// TwinCAT 3 PLC project PLC
// ProgramVersion: 3.1.4024.0
// libraries:
//   Tc2_DMX, * (Beckhoff Automation GmbH)
//   Tc2_EtherCAT, * (Beckhoff Automation GmbH)
//   Tc2_Standard, * (Beckhoff Automation GmbH)
//   Tc2_System, * (Beckhoff Automation GmbH)
//   Tc2_Utilities, * (Beckhoff Automation GmbH)
//   Tc3_Module, * (Beckhoff Automation GmbH)
//   VisuDialogs, * (System)
// project tree:
//   / GlobalTextList.TcGTLO, PlcTask.TcTTO, Visualisierungsmanager.TcVMO (not stored), VISU_TASK.TcTTO
//   POUs/ FBiFilter.TcPOU, iGetNextBufferPointer.TcPOU, iGetPriorBufferPointer.TcPOU, MAIN.TcPOU
//   VISUs/ Visu.TcVIS, Visualization.TcVIS (excluded from build)
// real-time tasks:
//   TASK PlcTask: cycle T#1ms, priority 20, ADS port 350
//   TASK VISU_TASK: cycle T#100000us, priority 30, ADS port 351
// I/O:
//   DEVICE Device 4 (EtherCAT), AmsNetId 192.168.0.150.5.1
//     Term 2 (EK1100) [EK1100 EtherCAT Coupler (2A E-Bus)]
//       Term 3 (EL6851) [EL6851 DMX Master]
//       Term 4 (EL9011) [EL9011 End Terminal]
//     Box 4 (EP3751-0260) [EP3751-0260 Acceleration Sensor]
// variable links:
//   PLC/PLC Instance <-> Device 4 (EtherCAT)/Box 4 (EP3751-0260)
//     PlcTask Inputs/MAIN.AccAxis[0] <-> AI Acc X Inputs/Value
//     PlcTask Inputs/MAIN.AccAxis[1] <-> AI Acc Y Inputs/Value
//     PlcTask Inputs/MAIN.AccAxis[2] <-> AI Acc Z Inputs/Value
//     PlcTask Inputs/MAIN.Axis[0] <-> AI Gyro X Inputs/Value
//     PlcTask Inputs/MAIN.Axis[1] <-> AI Gyro Y Inputs/Value
//     PlcTask Inputs/MAIN.Axis[2] <-> AI Gyro Z Inputs/Value
//     PlcTask Inputs/MAIN.ECATState <-> InfoData/State
//     PlcTask Inputs/MAIN.EcatPort <-> InfoData/AdsAddr/port
//     PlcTask Inputs/MAIN.dNetID <-> InfoData/AdsAddr/netId
//   PLC/PLC Instance <-> Device 4 (EtherCAT)/Term 2 (EK1100)/Term 3 (EL6851)
//     PlcTask Inputs/MAIN.stEL6851InData/bCyclicTxDDisabled <-> DMX Status/Cyclic TxD disabled
//     PlcTask Inputs/MAIN.stEL6851InData/bDefaultDataSent <-> DMX Status/Default data sent
//     PlcTask Inputs/MAIN.stEL6851InData/bFrameSentToggle <-> DMX Status/Frame sent toggle
//     PlcTask Inputs/MAIN.stEL6851InData/bInputToggle <-> WcState/InputToggle
//     PlcTask Inputs/MAIN.stEL6851InData/bReceiveToggle <-> DMX Status/Receive toggle
//     PlcTask Inputs/MAIN.stEL6851InData/bTransmitAccepted <-> DMX Status/Transmit accepted
//     PlcTask Inputs/MAIN.stEL6851InData/bTxPDOToggle <-> DMX Status/TxPDO Toggle
//     PlcTask Inputs/MAIN.stEL6851InData/bWcState <-> WcState/WcState
//     PlcTask Inputs/MAIN.stEL6851InData/byStartCode <-> DMX Status/Start code
//     PlcTask Inputs/MAIN.stEL6851InData/stAdsAddr <-> InfoData/AdsAddr
//     PlcTask Inputs/MAIN.stEL6851InData/uiState <-> InfoData/State
//     PlcTask Inputs/MAIN.stEL6851InData/wChannelLength <-> DMX Status/Channel length
//     PlcTask Outputs/MAIN.stEL6851OutData/arrData[{1..20}] <-> DMX Channel 1-64/Channel {1..20}  (20 links)
//     PlcTask Outputs/MAIN.stEL6851OutData/bDisableCyclicTxD <-> DMX Control/Disable cyclic TxD
//     PlcTask Outputs/MAIN.stEL6851OutData/bSendDefaultData <-> DMX Control/Send default data
//     PlcTask Outputs/MAIN.stEL6851OutData/bTransmitRequest <-> DMX Control/Transmit request
//     PlcTask Outputs/MAIN.stEL6851OutData/byStartCode <-> DMX Control/Start code
//     PlcTask Outputs/MAIN.stEL6851OutData/wChannelLength <-> DMX Control/Channel length

CONFIGURATION PLC
    RESOURCE PLC ON TwinCAT3
        TASK PlcTask(INTERVAL := T#1ms, PRIORITY := 20);
        TASK VISU_TASK(INTERVAL := T#100000us, PRIORITY := 30);
        PROGRAM MAIN WITH PlcTask : MAIN;
        PROGRAM VisuElems_Visu_Prg WITH VISU_TASK : VisuElems.Visu_Prg;
    END_RESOURCE
END_CONFIGURATION

// ---- POUs/MAIN.TcPOU
PROGRAM MAIN
VAR
(* Slave Information *)
	ECATState AT %I* : WORD;
	EcatPort AT %I* : WORD;
	netId : STRING(23);
	dNetID AT %I* : ARRAY [0..5] OF BYTE;

	Axis AT %I* : ARRAY [0..2] OF DINT;
	corrAxis : ARRAY [0..2] OF DINT;
	offset : ARRAY [0..2] OF DINT;

	Integrator : ARRAY [0..2] OF LREAL;
	Deg : ARRAY [0..2] OF LREAL;
	DegMovingHead : ARRAY [0..2] OF INT;
	z: INT;

	iFltValue : ARRAY [0..2] OF DINT;
	iFilter : ARRAY [0..2] OF FBiFilter;
	aFltArray : ARRAY [0..2] OF ARRAY [0..10000] OF DINT;
	
(* Accelerometer values *)
	AccAxis AT %I* : ARRAY [0..2] OF DINT;
	normalizedAcceleration : ARRAY [0..2] OF LREAL;

(* CoE Access *)
	WrCoe : FB_EcCoESdoWrite;
	RdCoe : FB_EcCoESdoRead;
	buf : POINTER TO INT;
	arBuf : ARRAY [0..5] OF BYTE;
	
(* Working variables *)
	slope : R_TRIG;
	bWriteOffset: BOOL;
	WriteOffsetState: INT;

	slopeResetCalibration : R_TRIG;
	bReset: BOOL;

	slopeResetAngle : R_TRIG;
	bResetAngle: BOOL;

	slopeReadFIFO : R_TRIG;
	bReadFIFO: BOOL;
	readFIFOState: INT;
	bytesToRead :INT := 1;
	rcvBytes : ARRAY [0..15] OF INT;
	bytesLeft: INT;
	
	dps : INT := 2000;
	
	(* state variables *)
	actualRoll : LREAL;
	actualPitch : LREAL;
	actualYaw : LREAL;
	
	actualPhi : LREAL;
	actualTheta : LREAL;
	actualGamma : LREAL;
		
	degPhi :INT;
	degTheta :INT;
	degGamma :INT;
	
	droll : LREAL;
	dpitch : LREAL;
	dyaw : LREAL;

	dphi : LREAL;
	dtheta : LREAL;
	dgamma : LREAL;

	temp : LREAL;
	
	AccPhi : LREAL;
	AccTheta : LREAL;
	
	sumAcc : LREAL;
	
	fusionWeight : LREAL := 1024;
	fusionWindow: INT := 50;
	fusionHorizontThreshold :LREAL := 0.4;


	//DMX
	stEL6851InData  AT%I*:  ST_EL6851InDataEx;
	stEL6851OutData AT%Q*: ST_EL6851OutData;
	stCommandBuffer : ST_DMXCommandBuffer;
	arrProcessData  : ARRAY [1..512] OF BYTE;
	
	fbDMX		: FB_EL6851CommunicationEx;
	aByte :array [1..2] of byte;
END_VAR

FOR z := 0 TO 2 DO
	(* Integrate the gyro values to gain an overall angle -> this angle is RPY *)
	corrAxis[z] := Axis[z] - offset[z];
	
	(* ignore values greater that +/-32000 *)
	IF corrAxis[z] > 32000 THEN corrAxis[z] := 0; END_IF;
	IF corrAxis[z] < -32000 THEN corrAxis[z] := 0; END_IF;

	Integrator[z] := Integrator[z] + (corrAxis[z] / (1000.0*(32768/dps)*90*4));
	Deg[z] := Integrator[z] * 360.0;
	DegMovingHead[z] := REAL_TO_INT(Deg[z]) MOD 360;

	(* Filter values for axis zero correction *)
	IF Axis[z] < 32000 AND Axis[z] > -32000 THEN
		iFilter[z](ptInputValue := ADR(Axis[z]), ptFilterArray := ADR(aFltArray[z]), iBufferSize := 2000, bExecute := 1);
		iFltValue[z] := iFilter[z].iFilterOutput;
	END_IF;
END_FOR

(* calculate the delta movements *)
droll := actualRoll;
dpitch := actualPitch;
dyaw := actualYaw;

actualRoll := (Deg[0] /360) * 2 * PI;
actualPitch := (Deg[1] /360) * 2 * PI;
actualYaw := (Deg[2] /360) * 2 * PI;

droll := actualRoll - droll;
dpitch := actualPitch - dpitch;
dyaw := actualYaw - dyaw;

(* Axis correction *)
dyaw := -dyaw;
temp := dpitch;
dpitch := droll;
droll := temp;

(* Calculate the euler speeds *)
dphi := droll + SIN(actualPhi)*TAN(actualTheta)*dpitch + COS(actualPhi)*TAN(actualTheta)*dyaw;
dtheta := COS(actualPhi)*dpitch-SIN(actualPhi)*dyaw;
dgamma := (SIN(actualPhi)/COS(actualTheta)) * dpitch + (COS(actualPhi)/COS(actualTheta)) * dyaw;

(* Calculate new euler angles *)
actualPhi := actualPhi + dphi;
actualTheta := actualTheta + dtheta;
actualGamma := actualGamma + dgamma;

(* Collapse if passing thresholds of pi *)
IF actualPhi < 0 THEN
	actualPhi := actualPhi + 2*PI;
END_IF
IF actualPhi >= 2*PI THEN
	actualPhi := actualPhi - 2*PI;
END_IF
IF actualTheta < 0 THEN
	actualTheta := actualTheta + 2*PI;
END_IF
IF actualTheta >= 2*PI THEN
	actualTheta := actualTheta - 2*PI;
END_IF
IF actualGamma < 0 THEN
	actualGamma := actualGamma + 2*PI;
END_IF
IF actualGamma >= 2*PI THEN
	actualGamma := actualGamma - 2*PI;
END_IF

(* Determine length of acceleration vector *)
sumAcc := AccAxis[0] * AccAxis[0] + AccAxis[1] * AccAxis[1] + AccAxis[2] * AccAxis[2];
sumAcc := SQRT(sumAcc);

(* Normalize acceleration vector *)
IF sumAcc <> 0 THEN
	FOR z := 0 TO 2 DO
		normalizedAcceleration[z] := AccAxis[z] / sumAcc;
	END_FOR
END_IF

(* Due to normalized values, we do no need to cut off higher values than 1 *)
IF normalizedAcceleration[2] = 0 THEN
	normalizedAcceleration[2] := 0.000001;
END_IF
AccPhi := -ATAN(normalizedAcceleration[0] / normalizedAcceleration[2]) + PI;
IF (AccAxis[2]) >=0 THEN
	AccPhi := AccPhi + PI;
END_IF
IF AccPhi > 2*PI THEN AccPhi := AccPhi - 2*PI; END_IF;
IF AccPhi < 0 THEN AccPhi := AccPhi + 2*PI; END_IF;
AccTheta := ASIN(normalizedAcceleration[1]) + PI;
(* Simple sensor fusion if we are not accelerated *)
IF sumAcc >= (2048 - fusionWindow) AND sumAcc <= (2048 + fusionWindow) THEN
	(* The AccPhi calculation is good, as long as Axis[2] ist not close to 0 *)
	IF normalizedAcceleration[2] < -fusionHorizontThreshold OR normalizedAcceleration[2] > fusionHorizontThreshold THEN
		IF (actualPhi - AccPhi) > PI OR (actualPhi - AccPhi) < -PI THEN
			IF AccPhi > actualPhi THEN
				AccPhi := AccPhi - 2 * PI;
			ELSE
				AccPhi := AccPhi + 2 * PI;
			END_IF
		END_IF
		actualPhi := ((fusionWeight-1) * actualPhi + AccPhi) /fusionWeight;
		(* error Zero crossing nicht beachtet!!! *)
	END_IF
	(* AccTheta is always accurate *)
	actualTheta := ((fusionWeight-1) * actualTheta + AccTheta) /fusionWeight;
END_IF

slope(CLK := bWriteOffset);
IF slope.Q THEN
	IF WriteOffsetState = 0 THEN
		WriteOffsetState := 0;
		FOR z := 0 TO 2 DO
			offset[z] := iFltValue[z];
			Integrator[z] := 0.5; 
		END_FOR
	END_IF;
END_IF

slopeResetCalibration(CLK := bReset);
IF slopeResetCalibration.Q THEN
	FOR z := 0 TO 2 DO
		offset[z] := 0;
		iFilter[z](bExecute := 0);
	END_FOR
END_IF

slopeResetAngle(CLK := bResetAngle);
IF slopeResetAngle.Q THEN
	FOR z := 0 TO 2 DO
		Integrator[z] := 0.5;
		actualRoll := PI;
		actualPitch := PI;
		actualYaw := PI;
		
		actualPhi := PI;
		actualTheta := PI;
		actualGamma := PI;
	END_FOR
END_IF

slopeReadFIFO(CLK := bReadFIFO);
IF slopeReadFIFO.Q THEN
	readFIFOState := 1;
	bytesLeft := bytesToRead;
END_IF

// calculation rad --> degree
degPhi 		:= TO_INT(actualPhi *360 /(2*PI));
degTheta	:= TO_INT(actualTheta *360 /(2*PI));
degGamma	:= TO_INT(actualGamma *360 /(2*PI));

DMX();

ACTION DMX:
//values depended on which box is used
//arrProcessData[1]:= TO_BYTE(LIMIT(0,(EP3751_0160_X*128/1100)+128,255));
//arrProcessData[2]:= TO_BYTE(LIMIT(0,(EP3751_0160_Y*128/1100)+128,255));

//arrProcessData[1]:= TO_BYTE(LIMIT(0,(EP3751_0260_X*128/1100)+128,255));
//arrProcessData[2]:= TO_BYTE(LIMIT(0,(EP3751_0260_rX*128/1100)+128,255));
//memcpy(ADR(aByte),ADR(corrAxis[2]),2);

arrProcessData[1]:= TO_BYTE(LIMIT(0,((actualGamma)*170/(2*PI)),255));
arrProcessData[2]:= TO_BYTE(LIMIT(0,((2*actualTheta-1.9*PI)*235/(2*PI)),255)); // 0..255
//arrProcessData[1]:=LIMIT(0,TO_BYTE(arrProcessData[1]+(-1*corrAxis[2]/1000)),255);
//arrProcessData[1]:=arrProcessData[1];
//arrProcessData[2]:=arrProcessData[2];
//static values
arrProcessData[3]:= 10;
arrProcessData[5]:= 255;
arrProcessData[6]:= 255;

fbDMX(
	wSourceManufacturerId:= 16#42_41, 
	dwSourceDeviceId:= 16#12_13_14_15, 
	bEnableSendingData:= TRUE, 
	bSetCycleMode:=TRUE , 
	bSendDefaultData:= , 
	uiDataLength:= 64 , 
	dwOptions:=  , 
	stEL6851InData:=	stEL6851InData , 
	stEL6851OutData:= 	stEL6851OutData, 
	stCommandBuffer:= 	stCommandBuffer, 
	arrProcessData:=	arrProcessData);
END_ACTION

END_PROGRAM

// ---- POUs/FBiFilter.TcPOU
FUNCTION_BLOCK FBiFilter
VAR_INPUT
	bExecute : BOOL;
	ptInputValue : POINTER TO INT;
	ptFilterArray : POINTER TO ARRAY [0..0] OF INT;
	iBufferSize: INT;
END_VAR
VAR_OUTPUT
	bRingbufferFilled : BOOL;
	iFilterOutput : INT;
END_VAR
VAR
	FilterSum : LREAL;
	iPtBufferPointer : INT;
	iValueCount : INT;
END_VAR

IF bExecute THEN
	FilterSum := FilterSum - ptFilterArray^[iPtBufferPointer];
	ptFilterArray^[iPtBufferPointer] := ptInputValue^;
	FilterSum := FilterSum + ptInputValue^;
	iPtBufferPointer := iGetNextBufferPointer(iBufferSize, iPtBufferPointer);
	iFilterOutput := LREAL_TO_INT(FilterSum / INT_TO_LREAL(iBufferSize));
	IF iValueCount >= iBufferSize THEN
		bRingbufferFilled := 1;
	ELSE
		iValueCount := iValueCount + 1;
	END_IF;
ELSE
	iValueCount := 0;
	bRingbufferFilled := 0;
END_IF;

END_FUNCTION_BLOCK

// ---- POUs/iGetNextBufferPointer.TcPOU
FUNCTION iGetNextBufferPointer : INT
VAR_INPUT
	iBufferSize : INT;
	iActualPointerValue : INT;
END_VAR
VAR
	retVal : INT;
END_VAR

retVal := iActualPointerValue + 1;
IF retVal >= iBufferSize THEN retVal := 0; END_IF;
iGetNextBufferPointer := retVal;

END_FUNCTION

// ---- POUs/iGetPriorBufferPointer.TcPOU
FUNCTION iGetPriorBufferPointer : INT
VAR_INPUT
	iBufferSize : INT;
	iActualPointerValue : INT;
END_VAR
VAR
	retVal : INT;
END_VAR

retVal := iActualPointerValue - 1;
IF retVal < 0 THEN retVal := iBufferSize - 1; END_IF;
iGetPriorBufferPointer := retVal;

END_FUNCTION

// ---- GlobalTextList.TcGTLO
TEXTLIST GlobalTextList
  216 = '%.3f'
  253 = '%d'
  686 = '%d°'
  671 = 'Abgleich'
  696 = 'Bytes: %d'
  952 = 'FThrh: %f'
  88 = 'FWeight: %f'
  277 = 'FWindow: %d'
  666 = 'Read FIFO'
  614 = 'Reset'
  479 = 'Reset Winkel'
END_TEXTLIST

// ---- VISUs/Visu.TcVIS
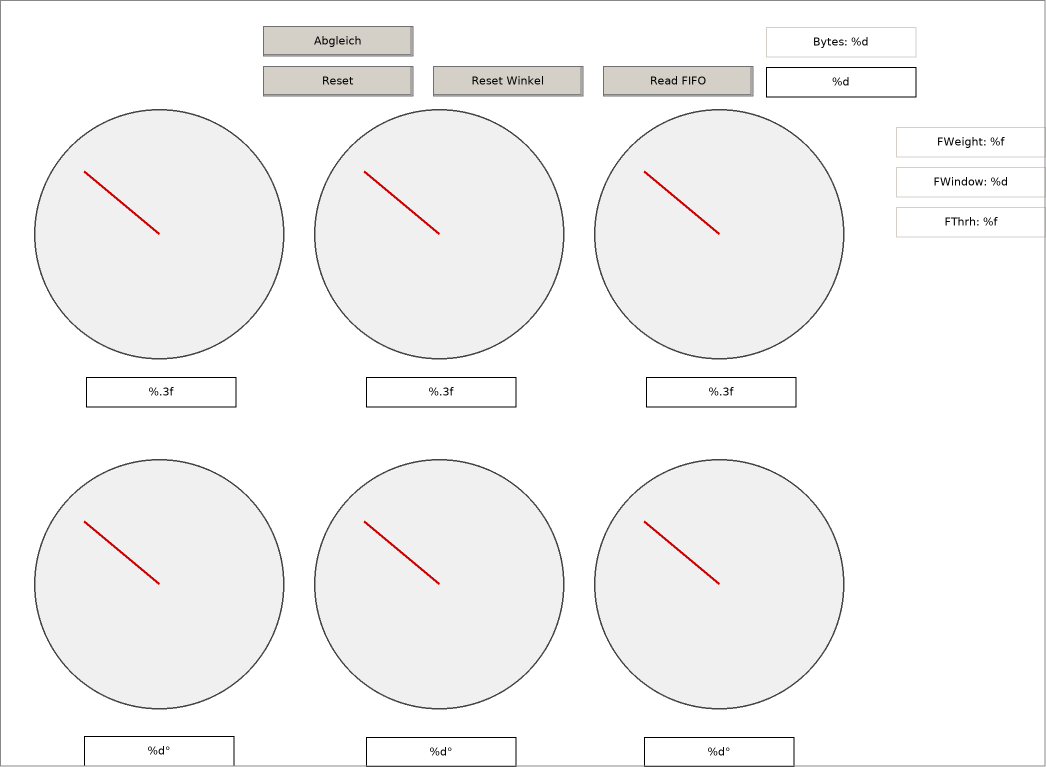
VISUALIZATION Visu  // 1046x767
    Meter360 (34,109 250x250), value: MAIN.DegMovingHead[2], style: Meter-Meter360-Gray, scale format: %d, scale 0..360
    Rectangle (86,377 150x30), "%.3f", text variable: MAIN.Deg[0]
    Button (263,26 150x30), "Abgleich", colour toggle: MAIN.iFilter[0].bRingbufferFilled
        p2175578022: 16#ffffff
        p573394764: 16#FFFF8080
        tap MAIN.bWriteOffset
    Button (263,66 150x30), "Reset"
        tap MAIN.bReset
    Meter360 (314,109 250x250), value: MAIN.DegMovingHead[1], style: Meter-Meter360-Gray, scale format: %d, scale 0..360
    Rectangle (366,377 150x30), "%.3f", text variable: MAIN.Deg[1]
    Meter360 (594,109 250x250), value: MAIN.DegMovingHead[0], style: Meter-Meter360-Gray, scale format: %d, scale 0..360
    Rectangle (646,377 150x30), "%.3f", text variable: MAIN.Deg[0]
    Button (433,66 150x30), "Reset Winkel"
        tap MAIN.bResetAngle
    Button (603,66 150x30), "Read FIFO"
        tap MAIN.bReadFIFO
    Rectangle (766,67 150x30), "%d", text variable: MAIN.arBuf[2]
    Textfield (766,27 150x30), "Bytes: %d", text variable: MAIN.bytesToRead
        OnMouseClick: write the text variable via Default
    Meter360 (34,459 250x250), value: MAIN.degGamma, style: Meter-Meter360-Gray, scale format: %d, scale 0..360
    Meter360 (314,459 250x250), value: MAIN.degTheta, style: Meter-Meter360-Gray, scale format: %d, scale 0..360
    Meter360 (594,459 250x250), value: MAIN.degPhi, style: Meter-Meter360-Gray, scale format: %d, scale 0..360
    Textfield (896,127 150x30), "FWeight: %f", text variable: MAIN.fusionWeight
        OnMouseClick: write the text variable via Default
    Textfield (896,167 150x30), "FWindow: %d", text variable: MAIN.fusionWindow
        OnMouseClick: write the text variable via Default
    Textfield (896,207 150x30), "FThrh: %f", text variable: MAIN.fusionHorizontThreshold
        OnMouseClick: write the text variable via Default
    Rectangle (84,736 150x30), "%d°", text variable: MAIN.degGamma
    Rectangle (366,737 150x30), "%d°", text variable: MAIN.degTheta
    Rectangle (644,737 150x30), "%d°", text variable: MAIN.degTheta
END_VISUALIZATION

// ---- VISUs/Visualization.TcVIS
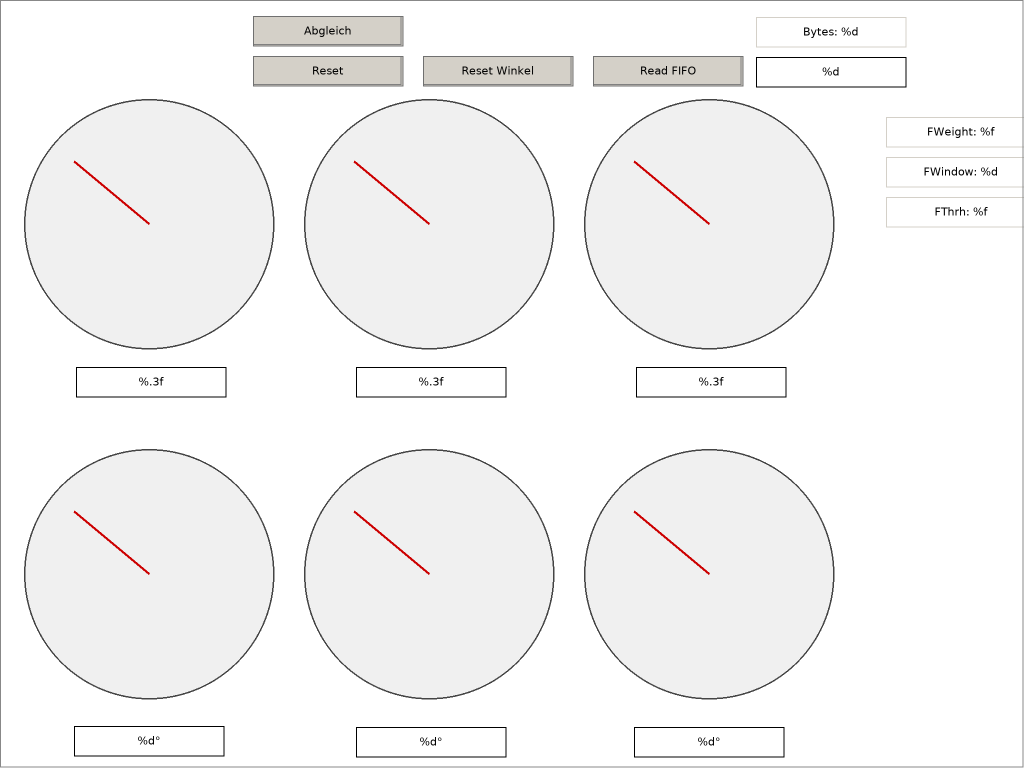
VISUALIZATION Visualization  // 1024x768
    Meter360 (24,99 250x250), value: MAIN.DegMovingHead[2], style: Meter-Meter360-Gray, scale format: %d, scale 0..360
    Rectangle (76,367 150x30), "%.3f", text variable: MAIN.Deg[0]
    Button (253,16 150x30), "Abgleich", colour toggle: MAIN.iFilter[0].bRingbufferFilled
        p2175578022: 16#ffffff
        p573394764: 16#FFFF8080
        tap MAIN.bWriteOffset
    Button (253,56 150x30), "Reset"
        tap MAIN.bReset
    Meter360 (304,99 250x250), value: MAIN.DegMovingHead[1], style: Meter-Meter360-Gray, scale format: %d, scale 0..360
    Rectangle (356,367 150x30), "%.3f", text variable: MAIN.Deg[1]
    Meter360 (584,99 250x250), value: MAIN.DegMovingHead[0], style: Meter-Meter360-Gray, scale format: %d, scale 0..360
    Rectangle (636,367 150x30), "%.3f", text variable: MAIN.Deg[0]
    Button (423,56 150x30), "Reset Winkel"
        tap MAIN.bResetAngle
    Button (593,56 150x30), "Read FIFO"
        tap MAIN.bReadFIFO
    Rectangle (756,57 150x30), "%d", text variable: MAIN.arBuf[2]
    Textfield (756,17 150x30), "Bytes: %d", text variable: MAIN.bytesToRead
        OnMouseClick: write the text variable via Default
    Meter360 (24,449 250x250), value: MAIN.degGamma, style: Meter-Meter360-Gray, scale format: %d, scale 0..360
    Meter360 (304,449 250x250), value: MAIN.degTheta, style: Meter-Meter360-Gray, scale format: %d, scale 0..360
    Meter360 (584,449 250x250), value: MAIN.degPhi, style: Meter-Meter360-Gray, scale format: %d, scale 0..360
    Textfield (886,117 150x30), "FWeight: %f", text variable: MAIN.fusionWeight
        OnMouseClick: write the text variable via Default
    Textfield (886,157 150x30), "FWindow: %d", text variable: MAIN.fusionWindow
        OnMouseClick: write the text variable via Default
    Textfield (886,197 150x30), "FThrh: %f", text variable: MAIN.fusionHorizontThreshold
        OnMouseClick: write the text variable via Default
    Rectangle (74,726 150x30), "%d°", text variable: MAIN.degGamma
    Rectangle (356,727 150x30), "%d°", text variable: MAIN.degTheta
    Rectangle (634,727 150x30), "%d°", text variable: MAIN.degTheta
END_VISUALIZATION
